RoboDK station: Project  zzz .rdk

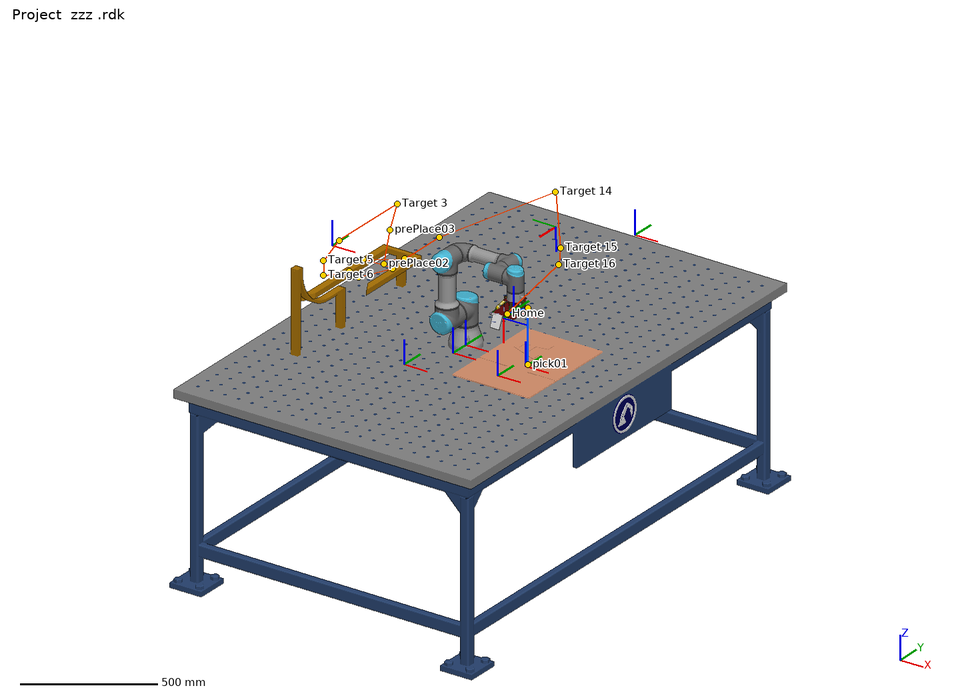
[picture v0: the station drawn from its stored meshes, robots at their saved joint values, targets as dots, program paths as lines]
Station Tast (saved by RoboDK 6.0.6). Poses are relative to the parent item; angles as X-Y-Z fixed-axis rotations.
  - frame Camera 1 at (420, -100, 590) mm, rotated rx -179.72 ry 0.28 rz -90 deg
    - camera Camera 1
  - frame Table at (20, -180, 0) mm
    - target Home (Cartesian target) at (261.4, -30.4, 243.15) mm, rotated rx -180 ry 0 rz -90 deg; joints [0, -90, -90, -90, 90, 0] of UR3
    - object Folding floor at (-460, -350, -50) mm, rotated rx 100 ry 0 rz -90 deg, size 300.1 x 350 x 30 mm, geometry from Folding floor.STEP
    - object  at (-530, -140, 140) mm, rotated rx 90 ry 0 rz -90 deg, size 530 x 140 x 167.7 mm, geometry from 2.STEP
    - object Table at (0, 800, 0) mm, rotated rx 0 ry 0 rz -90 deg, size 2020 x 1340 x 800 mm, geometry from Table-2000x1200x800mm.sld
  - frame UR3 Base at (20, -100, 0) mm
    - robot UR3: 6 axes, payload 3 kg, reach 500 mm, repeatability 0.1 mm, weight 11 kg
        modified DH rows (alpha deg, a mm, theta deg, d mm): 0, 0, 0, 151.9; 90, 0, 180, 0; 0, 243.65, 0, 0; 0, 213, 0, 110.4; -90, 0, 0, 83.4; 90, 0, 180, 82.4
        joint limits [-360, -360, -360, -360, -360, -360] to [360, 360, 360, 360, 360, 360]; home [0, -90, -90, 0, 90, 0]; saved at [0, -90, -90, -90, 90, 0]
      - tool VaccumTool, TCP at (0, 35, 70) mm, size 142.5 x 102 x 100.1 mm, geometry from Assem1.STEP
  - frame off_Box at (0, 230, 0) mm
  - frame Orinal_Box at (300, -120, 0) mm
    - target prepick01 (Cartesian target) at (10, 0, 240) mm, rotated rx 180 ry 0 rz -90 deg; joints [16.298, -92.34, -88.452, -89.208, 90, 16.298] of UR3
    - target pick01 (Cartesian target) at (10, 0, 10) mm, rotated rx 180 ry 0 rz -90 deg; joints [16.298, -123.225, -121.951, -24.825, 90, 16.298] of UR3
    - object BOX at (-32.54, 5.23, 0) mm, rotated rx 90 ry 0 rz 90 deg, size 470 x 7 x 340 mm, geometry from BOX.STEP
  - frame Frame 6 at (260, -240, 0) mm
  - frame Orinal_Box(2) at (-70, -360, 0) mm
    - target prePlace02 (Cartesian target) at (-17.01, -105.4, 444.11) mm, rotated rx -90 ry 5.56 rz -180 deg; joints [-90, -90, -90, 0, 90, 5.56] of UR3
    - target prePlace03 (Cartesian target) at (-17.01, -66.75, 566.16) mm, rotated rx -69.91 ry 5.22 rz -178.09 deg; joints [-90, -90, -70, 0, 90, 5.56] of UR3
    - target Target 3 (Cartesian target) at (-290, 370.4, 420.59) mm, rotated rx -90.01 ry 0 rz 90 deg; joints [-180, -93.722, -92.427, 6.14, 89.999, 0] of UR3
    - target Target 4 (Cartesian target) at (-290, 0.4, 420.59) mm, rotated rx -90.01 ry 0 rz 90 deg; joints [-112.594, -117.936, -60.702, -1.387, 22.593, 0.023] of UR3
    - target Target 5 (Cartesian target) at (-290.02, -99.93, 378.06) mm, rotated rx -90.03 ry 59.99 rz 89.98 deg; joints [-108.63, -135.02, -48.19, 3.17, 18.63, 60.03] of UR3
    - target Target 6 (Cartesian target) at (-290.02, -99.93, 318.06) mm, rotated rx -90.03 ry 59.99 rz 89.98 deg; joints [-108.63, -138.103, -58.934, 16.998, 18.63, 60.029] of UR3
    - target Target 7 (Cartesian target) at (-280, 50.05, 278.08) mm, rotated rx -90.02 ry 59.99 rz 89.98 deg; joints [-117.428, -117.824, -108.935, 46.732, 27.428, 60.014] of UR3
    - target Target 8 (Cartesian target) at (-280.01, 80.05, 248.08) mm, rotated rx -90.02 ry 59.99 rz 89.98 deg; joints [-120.775, -120.746, -116.476, 57.199, 30.775, 60.011] of UR3
    - target Target 9 (Cartesian target) at (-280.01, 110.39, 230.55) mm, rotated rx -90.02 ry -0.02 rz 90 deg; joints [-120.78, -120.75, -116.48, 57.2, 30.78, 0.01] of UR3
    - target Target 10 (Cartesian target) at (-220.01, 240.39, 230.55) mm, rotated rx -90.02 ry -0.02 rz 90 deg; joints [-128.874, -104.188, -151.003, 75.166, 38.874, 0.004] of UR3
    - target Target 11 (Cartesian target) at (-350.01, 240.39, 230.55) mm, rotated rx -90.02 ry -0.02 rz 90 deg; joints [-153.581, -124.593, -108.484, 53.059, 63.581, -0.008] of UR3
    - target Target 12 (Cartesian target) at (-230.01, 330.39, 230.55) mm, rotated rx -90.02 ry -0.02 rz 90 deg; joints [-165.384, -107.985, -143.061, 71.03, 75.384, -0.012] of UR3
    - target Target 13 (Cartesian target) at (-230.01, 550.39, 230.55) mm, rotated rx -90.02 ry -0.02 rz 90 deg; joints [-220.78, -132.513, -91.991, 44.484, 130.78, -0.029] of UR3
    - target Target 14 (Cartesian target) at (190.11, 686.48, 476.9) mm, rotated rx -90.03 ry -0.03 rz 0 deg; joints [-267.83, -104.5, -64.46, -11.07, 87.83, -0.03] of UR3
    - target Target 15 (Cartesian target) at (237.66, 648.87, 277.57) mm, rotated rx 177.83 ry 0.03 rz 92.2 deg; joints [-269.487, -113.384, -52.223, -104.36, 87.83, -91.688] of UR3
    - target Target 16 (Cartesian target) at (231.95, 647.78, 210) mm, rotated rx -180 ry -0.03 rz 90.51 deg; joints [-269.49, -111.831, -72.402, -85.737, 90, -90] of UR3
  - Python program main (listed below)
  - Python program ClosedBox (listed below)
  - Python program ClosedBox2 (listed below)
  - Python program RE_BOX (listed below)
  - program pick (11 instructions, listed below)
  - program Place (24 instructions, listed below)
  - frame VaccumTool_Init at (0, 1000, 0) mm
    - object Box 215x215mm (Fold 2) at (0, 0, 0) mm, size 213.4 x 213.4 x 444 mm, geometry from Box-215x215mm-Fold-2.sld
  - frame VaccumTool_Ref at (300, -260, 250) mm, rotated rx 0 ry 90 rz 0 deg
  - frame Vaccum_Init at (0, 1000, 0) mm
    - object Box 215x215mm (Fold 3) at (0, 0, 0) mm, size 213.4 x 213.4 x 346.2 mm, geometry from Box-215x215mm-Fold-3.sld
  - frame Vaccum_Ref at (-510, -190, 290) mm
  - program RE (1 instructions, listed below)
  - program RUN (2 instructions, listed below)
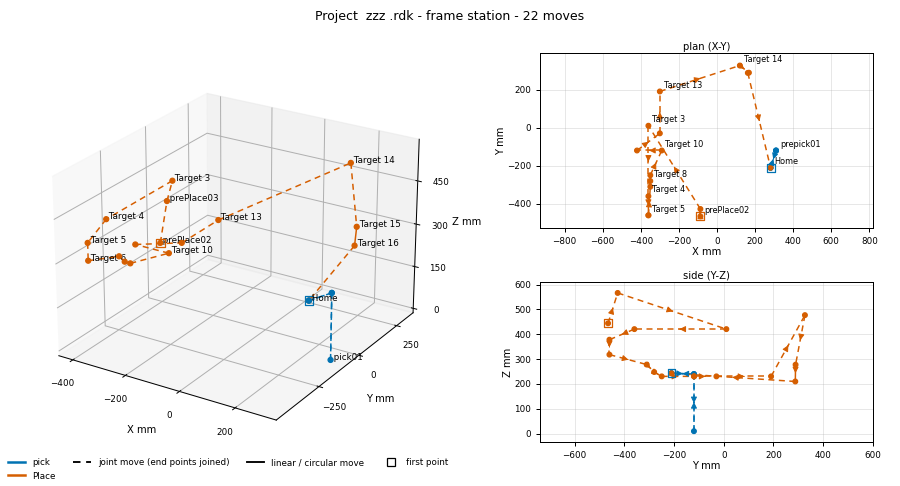
[picture p0: tool path of Project  zzz .rdk in frame station, 22 of 22 moves have a stored position in this frame; points joined in program order, loops and branches not executed]

--- Python program main ---
# Type help("robodk.robolink") or help("robodk.robomath") for more information
# Press F5 to run the script
# Documentation: https://robodk.com/doc/en/RoboDK-API.html
# Reference:     https://robodk.com/doc/en/PythonAPI/robodk.html
# Note: It is not required to keep a copy of this file, your Python script is saved with your RDK project

# You can also use the new version of the API:
from robodk import robolink    # RoboDK API
from robodk import robomath    # Robot toolbox
RDK = robolink.Robolink()

# Forward and backwards compatible use of the RoboDK API:
# Remove these 2 lines to follow python programming guidelines
from robodk import *      # RoboDK API
from robolink import *    # Robot toolbox
# Link to RoboDK
# RDK = Robolink()

# Notify user:
print('To edit this program:\nright click on the Python program, then, select "Edit Python script"')

# Program example:
item = RDK.Item('base')
if item.Valid():
    print('Item selected: ' + item.Name())
    print('Item posistion: ' + repr(item.Pose()))

print('Items in the station:')
itemlist = RDK.ItemList()
print(itemlist)

# Provoking an exception will display the console output if you run this script from RoboDK
raise Exception('Program not edited.')

--- Python program ClosedBox ---
# Type help("robolink") or help("robodk") for more information
# Press F5 to run the script
# Documentation: https://robodk.com/doc/en/RoboDK-API.html
# Reference:     https://robodk.com/doc/en/PythonAPI/index.html
# Note: It is not required to keep a copy of this file, your python script is saved with the station
from robodk import robolink

RDK = robolink.Robolink()

#----- Constante -----

NEW_OBJECT_NAME = 'ClosedBox' #Name of the new object created
REFERENCE_FRAME_INIT = 'VaccumTool_Init'
REFERENCE_FRAME_REF = "VaccumTool_Ref"
REF_TOOL = "VaccumTool"



#------- Program ------
frame_init = RDK.Item(REFERENCE_FRAME_INIT, robolink.ITEM_TYPE_FRAME)
frame_ref = RDK.Item(REFERENCE_FRAME_REF, robolink.ITEM_TYPE_FRAME)
tool = RDK.Item(REF_TOOL, robolink.ITEM_TYPE_TOOL)

RDK.Render(False)

for item in tool.Childs():
    if item.Type() == robolink.ITEM_TYPE_OBJECT:
        item.setVisible(False)

if frame_ref.Valid():
    for item in frame_init.Childs():
        item.Copy()
        new_obj = RDK.Paste()
        new_obj.setVisible(False)
        new_obj.setParent(frame_ref)
        new_obj.setName(NEW_OBJECT_NAME)
        RDK.Update()
        new_obj.setParentStatic(tool)
        new_obj.setVisible(True)

RDK.Render(True)

--- Python program ClosedBox2 ---
from robolink import *
from robodk import *

RDK = Robolink()

# =========================================================
# CONSTANT
# =========================================================

NEW_OBJECT_NAME = 'ClosedBox2'

REFERENCE_FRAME_INIT = 'Vaccum_Init'
REFERENCE_FRAME_REF  = 'Vaccum_Ref'
REF_TOOL = 'VaccumTool'


# =========================================================
# FIND ITEMS
# =========================================================

frame_init = RDK.Item(
    REFERENCE_FRAME_INIT,
    ITEM_TYPE_FRAME
)

frame_ref = RDK.Item(
    REFERENCE_FRAME_REF,
    ITEM_TYPE_FRAME
)

tool = RDK.Item(
    REF_TOOL,
    ITEM_TYPE_TOOL
)


# =========================================================
# CHECK
# =========================================================

if not frame_init.Valid():
    raise Exception("ไม่พบ Frame: Vaccum_Init")

if not frame_ref.Valid():
    raise Exception("ไม่พบ Frame: Vaccum_Ref")

if not tool.Valid():
    raise Exception("ไม่พบ Tool: VaccumTool")


# =========================================================
# START
# =========================================================

RDK.Render(False)

print("================================")
print("เริ่มเปลี่ยนวัตถุ")
print("================================")


# =========================================================
# 1. ซ่อนวัตถุเก่าที่อยู่กับ VaccumTool
# =========================================================

print("กำลังซ่อนวัตถุเก่า...")

for old_item in tool.Childs():

    if old_item.Type() == ITEM_TYPE_OBJECT:

        print(
            "ซ่อน:",
            old_item.Name()
        )

        # ซ่อนเท่านั้น ไม่ลบ
        old_item.setVisible(False)


# =========================================================
# 2. Copy วัตถุใหม่จาก Vaccum_Init
# =========================================================

print("กำลังสร้างวัตถุใหม่...")

for item in frame_init.Childs():

    if item.Type() != ITEM_TYPE_OBJECT:
        continue

    print(
        "Copy:",
        item.Name()
    )

    item.Copy()

    new_obj = RDK.Paste()

    if not new_obj.Valid():
        print("ERROR: สร้างวัตถุใหม่ไม่สำเร็จ")
        continue


    # =====================================================
    # 3. ซ่อนวัตถุใหม่ก่อน
    # =====================================================

    new_obj.setVisible(False)


    # =====================================================
    # 4. ตั้ง Parent
    # =====================================================

    new_obj.setParent(frame_ref)


    # =====================================================
    # 5. ตั้งชื่อ
    # =====================================================

    new_obj.setName(
        NEW_OBJECT_NAME
    )

    RDK.Update()


    # =====================================================
    # 6. ติดวัตถุใหม่กับ VaccumTool
    # =====================================================

    new_obj.setParentStatic(tool)


    # =====================================================
    # 7. แสดงวัตถุใหม่
    # =====================================================

    new_obj.setVisible(True)

    print(
        "แสดงวัตถุใหม่:",
        NEW_OBJECT_NAME
    )


# =========================================================
# FINISH
# =========================================================

RDK.Render(True)

print("================================")
print("เสร็จเรียบร้อย")
print("วัตถุเก่า = ซ่อน")
print("วัตถุใหม่ = แสดง")
print("================================")

--- Python program RE_BOX ---
from robodk.robolink import *
from robodk.robomath import *
import time

# =========================================================
# CONNECT ROBODK
# =========================================================

RDK = Robolink()


# =========================================================
# GET FRAME
# =========================================================

original_box = RDK.Item('Orinal_Box', ITEM_TYPE_FRAME)

if not original_box.Valid():
    raise Exception("ไม่พบ Frame: Orinal_Box")


# =========================================================
# GET BOX
# =========================================================

box = RDK.Item('BOX', ITEM_TYPE_OBJECT)

if not box.Valid():
    raise Exception("ไม่พบ Object: BOX")


# =========================================================
# ตำแหน่ง BOX ตอนเริ่มต้น
#
# อ้างอิงจากรูปของคุณ
#
# X  = -32.537
# Y  =   5.232
# Z  =   0
#
# Rotation
# X = 90
# Y = 0
# Z = 90
# =========================================================

BOX_HOME = transl(
    -32.537,
     5.232,
     0.000
)

# =========================================================
# ROTATION
# =========================================================
#
# ใช้ลำดับ Z -> Y -> X
# เพื่อให้ BOX นอนเหมือนตำแหน่งใน RoboDK
#

BOX_HOME = BOX_HOME \
    * rotz(90 * pi / 180) \
    * roty(0 * pi / 180) \
    * rotx(90 * pi / 180)


# =========================================================
# RESET BOX
# =========================================================

def reset_box():

    print("================================")
    print("RESET BOX")
    print("================================")

    # กลับตำแหน่งเดิม
    box.setPose(BOX_HOME)

    # แสดง BOX
    box.setVisible(True)

    # รอ RoboDK
    time.sleep(0.2)

    print("BOX RESET แล้ว")
    print("BOX แสดงแล้ว")
    print("================================")


# =========================================================
# HIDE BOX
# =========================================================

def hide_box():

    box.setVisible(False)

    print("BOX ถูกซ่อน")


# =========================================================
# SHOW BOX
# =========================================================

def show_box():

    box.setVisible(True)

    print("BOX แสดงแล้ว")


# =========================================================
# MAIN
# =========================================================

if __name__ == "__main__":

    reset_box()

--- program pick (robot UR3) ---
  Set Ref.: Table
  Set Tool: VaccumTool
  MoveL (Home)
  Set Ref.: Orinal_Box
  MoveJ (prepick01)
  MoveJ (pick01)
  Attach to VaccumTool
  MoveJ (prepick01)
  Set Ref.: Table
  MoveJ (Home)
  Call ClosedBox

--- program Place (robot UR3) ---
  Set Ref.: Orinal_Box(2)
  Set Tool: VaccumTool
  MoveJ (prePlace02)
  MoveJ (prePlace03)
  MoveJ (Target 3)
  MoveJ (Target 4)
  MoveJ (Target 5)
  MoveJ (Target 6)
  MoveJ (Target 7)
  MoveJ (Target 8)
  MoveJ (Target 9)
  MoveJ (Target 10)
  MoveJ (Target 11)
  MoveJ (Target 12)
  โทร ClosedBox2
  MoveJ (Target 13)
  MoveJ (Target 14)
  MoveJ (Target 15)
  MoveL (Target 16)
  Detach from VaccumTool
  Set Ref.: Table
  MoveJ (Home)
  Call RE
  Call RE_BOX

--- program RE (robot UR3) ---
  Move BOX

--- program RUN (robot UR3) ---
  Call pick
  Call Place
